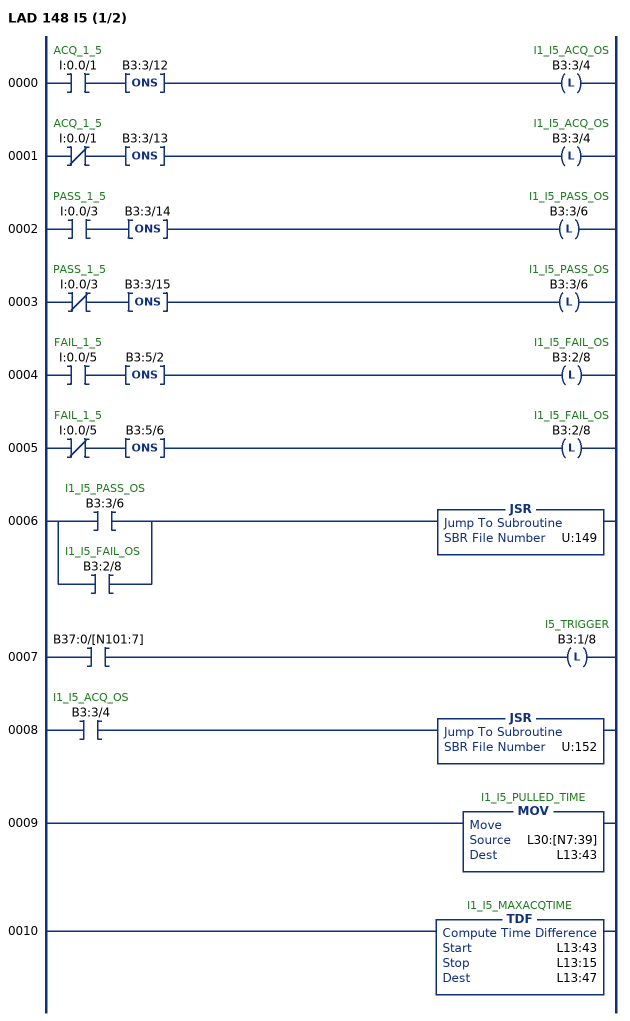
% Rung: 0 %
SOR XIC I:0.0/1 ONS B3:3/12 OTL B3:3/4 EOR
%   I:0.0/1  ACQ_1_5 %
%   B3:3/4  I1_I5_ACQ_OS %
% Rung: 1 %
SOR XIO I:0.0/1 ONS B3:3/13 OTL B3:3/4 EOR
%   I:0.0/1  ACQ_1_5 %
%   B3:3/4  I1_I5_ACQ_OS %
% Rung: 2 %
SOR XIC I:0.0/3 ONS B3:3/14 OTL B3:3/6 EOR
%   I:0.0/3  PASS_1_5 %
%   B3:3/6  I1_I5_PASS_OS %
% Rung: 3 %
SOR XIO I:0.0/3 ONS B3:3/15 OTL B3:3/6 EOR
%   I:0.0/3  PASS_1_5 %
%   B3:3/6  I1_I5_PASS_OS %
% Rung: 4 %
SOR XIC I:0.0/5 ONS B3:5/2 OTL B3:2/8 EOR
%   I:0.0/5  FAIL_1_5 %
%   B3:2/8  I1_I5_FAIL_OS %
% Rung: 5 %
SOR XIO I:0.0/5 ONS B3:5/6 OTL B3:2/8 EOR
%   I:0.0/5  FAIL_1_5 %
%   B3:2/8  I1_I5_FAIL_OS %
% Rung: 6 %
SOR BST XIC B3:3/6 NXB XIC B3:2/8 BND JSR U:149 EOR
%   B3:3/6  I1_I5_PASS_OS %
%   B3:2/8  I1_I5_FAIL_OS %
% Rung: 7 %
SOR XIC B37:0/[N101:7] OTL B3:1/8 EOR
%   B37:0  TOP_OK_1 %
%   N101:7  I5_TRIG_LOC %
%   B3:1/8  I5_TRIGGER %
% Rung: 8 %
SOR XIC B3:3/4 JSR U:152 EOR
%   B3:3/4  I1_I5_ACQ_OS %
% Rung: 9 %
SOR MOV L30:[N7:39] L13:43 EOR
%   N7:39  I5_OLDEST_PART_INDEX %
%   L13:43  I1_I5_PULLED_TIME %
% Rung: 10 %
SOR TDF L13:43 L13:15 L13:47 EOR
%   L13:43  I1_I5_PULLED_TIME %
%   L13:15  THE_TIME %
%   L13:47  I1_I5_MAXACQTIME %

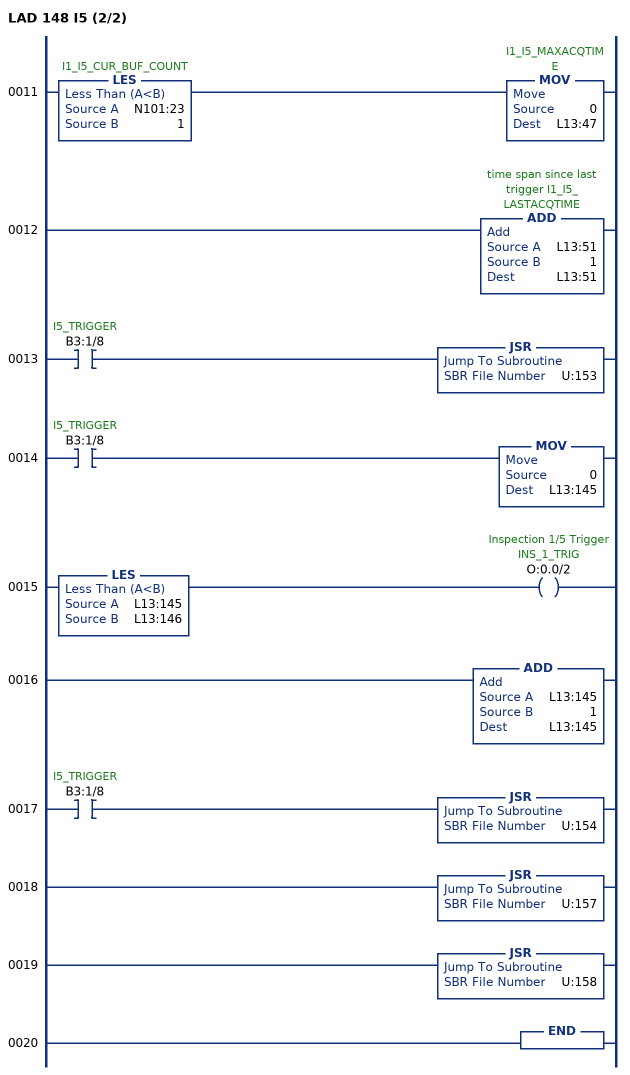
% Rung: 11 %
SOR LES N101:23 1 MOV 0 L13:47 EOR
%   N101:23  I1_I5_CUR_BUF_COUNT %
%   L13:47  I1_I5_MAXACQTIME %
% Rung: 12 %
SOR ADD L13:51 1 L13:51 EOR
%   L13:51  I1_I5_LASTACQTIME  "time span since last trigger" %
% Rung: 13 %
SOR XIC B3:1/8 JSR U:153 EOR
%   B3:1/8  I5_TRIGGER %
% Rung: 14 %
SOR XIC B3:1/8 MOV 0 L13:145 EOR
%   B3:1/8  I5_TRIGGER %
% Rung: 15 %
SOR LES L13:145 L13:146 OTE O:0.0/2 EOR
%   O:0.0/2  INS_1_TRIG  "Inspection 1/5 Trigger" %
% Rung: 16 %
SOR ADD L13:145 1 L13:145 EOR
% Rung: 17 %
SOR XIC B3:1/8 JSR U:154 EOR
%   B3:1/8  I5_TRIGGER %
% Rung: 18 %
SOR JSR U:157 EOR
% Rung: 19 %
SOR JSR U:158 EOR
% Rung: 20 %
SOR END EOR

LADDER 149 "I5 RESULT"
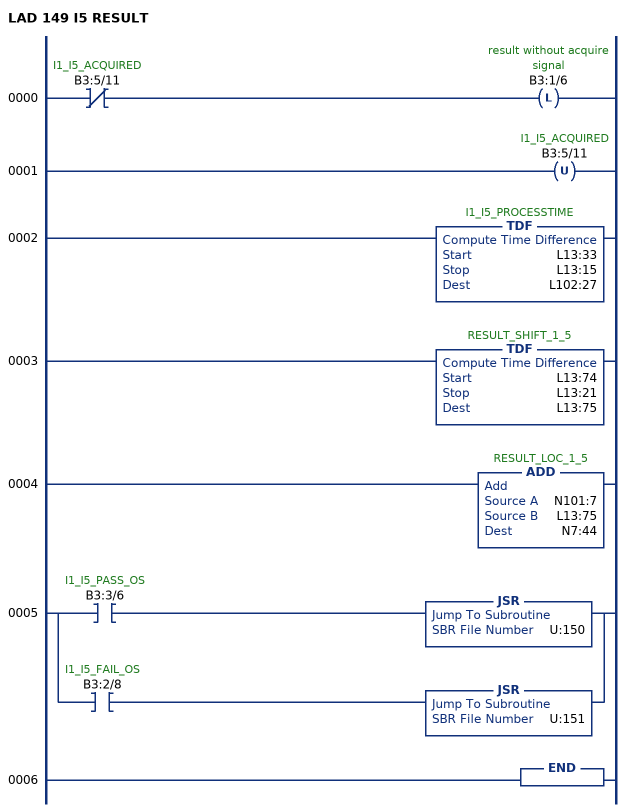
% Rung: 0 %
SOR XIO B3:5/11 OTL B3:1/6 EOR
%   B3:5/11  I1_I5_ACQUIRED %
%   B3:1/6  "result without acquire signal" %
% Rung: 1 %
SOR OTU B3:5/11 EOR
%   B3:5/11  I1_I5_ACQUIRED %
% Rung: 2 %
SOR TDF L13:33 L13:15 L102:27 EOR
%   L13:33  I1_I5_TIMEOFACQ %
%   L13:15  THE_TIME %
%   L102:27  I1_I5_PROCESSTIME %
% Rung: 3 %
SOR TDF L13:74 L13:21 L13:75 EOR
%   L13:74  I1_I5_PROC_START_POS %
%   L13:21  TOP_POSITION %
%   L13:75  RESULT_SHIFT_1_5 %
% Rung: 4 %
SOR ADD N101:7 L13:75 N7:44 EOR
%   N101:7  I5_TRIG_LOC %
%   L13:75  RESULT_SHIFT_1_5 %
%   N7:44  RESULT_LOC_1_5 %
% Rung: 5 %
SOR BST XIC B3:3/6 JSR U:150 NXB XIC B3:2/8 JSR U:151 BND EOR
%   B3:3/6  I1_I5_PASS_OS %
%   B3:2/8  I1_I5_FAIL_OS %
% Rung: 6 %
SOR END EOR

LADDER 150 "I5 PASS"
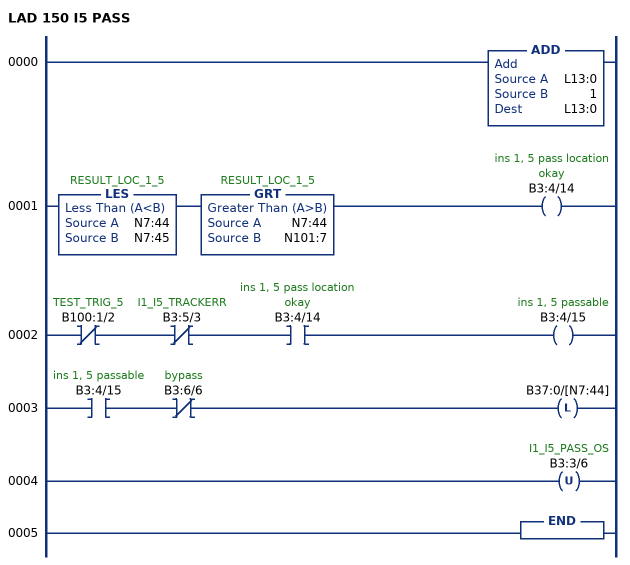
% Rung: 0 %
SOR ADD L13:0 1 L13:0 EOR
% Rung: 1 %
SOR LES N7:44 N7:45 GRT N7:44 N101:7 OTE B3:4/14 EOR
%   N7:44  RESULT_LOC_1_5 %
%   N7:45  I5_MAX_SHIFT  "ins 5 maximum result location" %
%   N101:7  I5_TRIG_LOC %
%   B3:4/14  "ins 1, 5 pass location okay" %
% Rung: 2 %
SOR XIO B100:1/2 XIO B3:5/3 XIC B3:4/14 OTE B3:4/15 EOR
%   B100:1/2  TEST_TRIG_5 %
%   B3:5/3  I1_I5_TRACKERR %
%   B3:4/14  "ins 1, 5 pass location okay" %
%   B3:4/15  "ins 1, 5 passable" %
% Rung: 3 %
SOR XIC B3:4/15 XIO B3:6/6 OTL B37:0/[N7:44] EOR
%   B3:4/15  "ins 1, 5 passable" %
%   B3:6/6  "bypass" %
%   B37:0  TOP_OK_1 %
%   N7:44  RESULT_LOC_1_5 %
% Rung: 4 %
SOR OTU B3:3/6 EOR
%   B3:3/6  I1_I5_PASS_OS %
% Rung: 5 %
SOR END EOR

LADDER 151 "I5 FAIL"
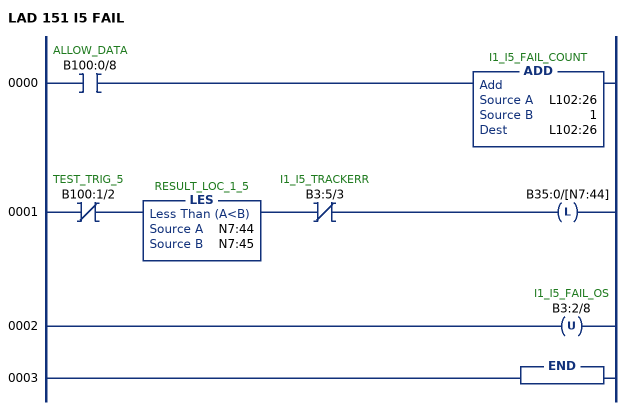
% Rung: 0 %
SOR XIC B100:0/8 ADD L102:26 1 L102:26 EOR
%   B100:0/8  ALLOW_DATA %
%   L102:26  I1_I5_FAIL_COUNT %
% Rung: 1 %
SOR XIO B100:1/2 LES N7:44 N7:45 XIO B3:5/3 OTL B35:0/[N7:44] EOR
%   B100:1/2  TEST_TRIG_5 %
%   N7:44  RESULT_LOC_1_5 %
%   N7:45  I5_MAX_SHIFT  "ins 5 maximum result location" %
%   B3:5/3  I1_I5_TRACKERR %
%   B35:0  TOP_NG %
% Rung: 2 %
SOR OTU B3:2/8 EOR
%   B3:2/8  I1_I5_FAIL_OS %
% Rung: 3 %
SOR END EOR

LADDER 152 "I5 ACQ"
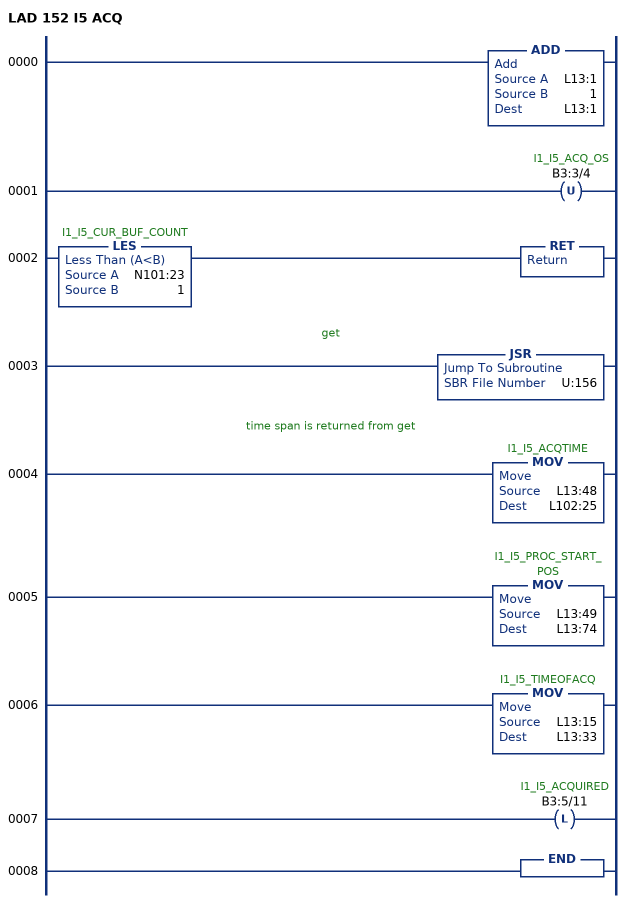
% Rung: 0 %
SOR ADD L13:1 1 L13:1 EOR
% Rung: 1 %
SOR OTU B3:3/4 EOR
%   B3:3/4  I1_I5_ACQ_OS %
% Rung: 2 %
SOR LES N101:23 1 RET EOR
%   N101:23  I1_I5_CUR_BUF_COUNT %
% Rung: 3 %
% get %
SOR JSR U:156 EOR
% Rung: 4 %
% time span is returned from get %
SOR MOV L13:48 L102:25 EOR
%   L13:48  I1_I5_TIME_SPAN %
%   L102:25  I1_I5_ACQTIME %
% Rung: 5 %
SOR MOV L13:49 L13:74 EOR
%   L13:49  I1_I5_PULLED_POS %
%   L13:74  I1_I5_PROC_START_POS %
% Rung: 6 %
SOR MOV L13:15 L13:33 EOR
%   L13:15  THE_TIME %
%   L13:33  I1_I5_TIMEOFACQ %
% Rung: 7 %
SOR OTL B3:5/11 EOR
%   B3:5/11  I1_I5_ACQUIRED %
% Rung: 8 %
SOR END EOR

LADDER 153 "I5 TESTER"
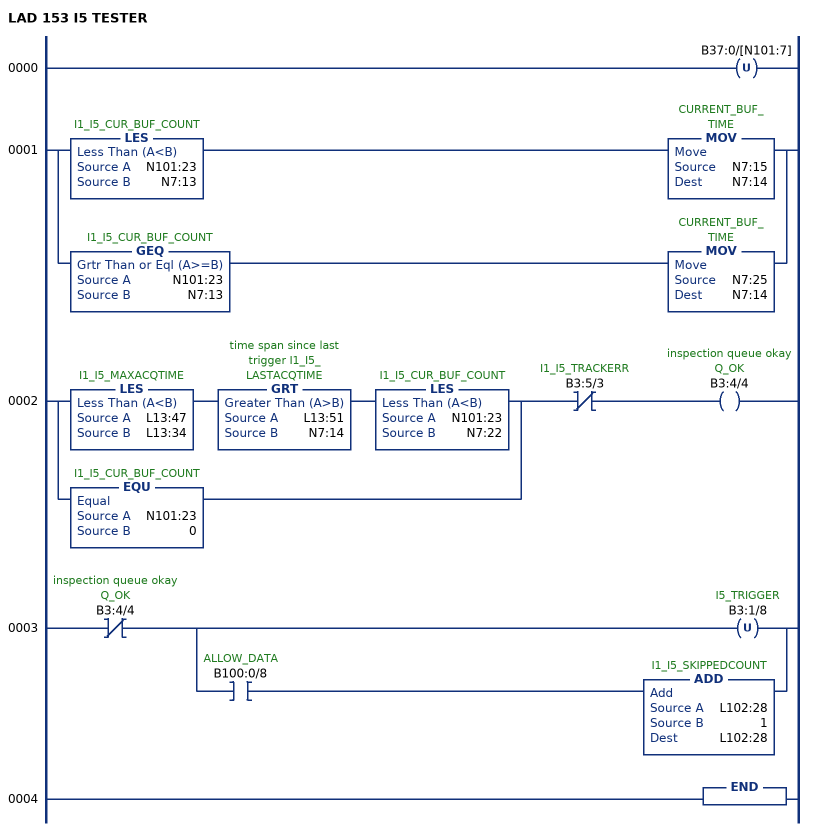
% Rung: 0 %
SOR OTU B37:0/[N101:7] EOR
%   B37:0  TOP_OK_1 %
%   N101:7  I5_TRIG_LOC %
% Rung: 1 %
SOR BST LES N101:23 N7:13 MOV N7:15 N7:14 NXB GEQ N101:23 N7:13 MOV N7:25 N7:14 BND EOR
%   N101:23  I1_I5_CUR_BUF_COUNT %
%   N7:13  BUF_TRANS  "cam to pc buf transition" %
%   N7:15  CAM_BUF_TIME  "cam buf time" %
%   N7:14  CURRENT_BUF_TIME %
%   N7:25  PC_BUF_TIME  "pc buf time" %
% Rung: 2 %
SOR BST LES L13:47 L13:34 GRT L13:51 N7:14 LES N101:23 N7:22 NXB EQU N101:23 0 BND XIO B3:5/3 OTE B3:4/4 EOR
%   L13:47  I1_I5_MAXACQTIME %
%   L13:34  MAX_ACQ_ALL  "absolute max acquire time before bypass trigger" %
%   L13:51  I1_I5_LASTACQTIME  "time span since last trigger" %
%   N7:14  CURRENT_BUF_TIME %
%   N101:23  I1_I5_CUR_BUF_COUNT %
%   N7:22  MAX_BUF_ALL  "max buffer count alowed before bypass" %
%   B3:5/3  I1_I5_TRACKERR %
%   B3:4/4  Q_OK  "inspection queue okay" %
% Rung: 3 %
SOR XIO B3:4/4 BST OTU B3:1/8 NXB XIC B100:0/8 ADD L102:28 1 L102:28 BND EOR
%   B3:4/4  Q_OK  "inspection queue okay" %
%   B3:1/8  I5_TRIGGER %
%   B100:0/8  ALLOW_DATA %
%   L102:28  I1_I5_SKIPPEDCOUNT %
% Rung: 4 %
SOR END EOR

LADDER 154 "I5 TRIG"
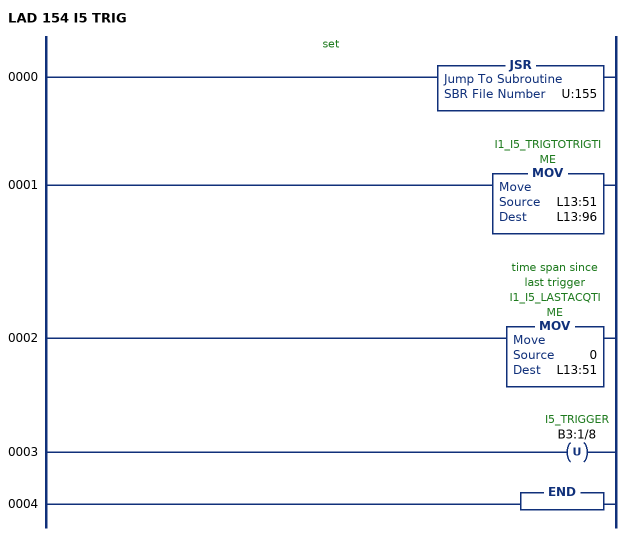
% Rung: 0 %
% set %
SOR JSR U:155 EOR
% Rung: 1 %
SOR MOV L13:51 L13:96 EOR
%   L13:51  I1_I5_LASTACQTIME  "time span since last trigger" %
%   L13:96  I1_I5_TRIGTOTRIGTIME %
% Rung: 2 %
SOR MOV 0 L13:51 EOR
%   L13:51  I1_I5_LASTACQTIME  "time span since last trigger" %
% Rung: 3 %
SOR OTU B3:1/8 EOR
%   B3:1/8  I5_TRIGGER %
% Rung: 4 %
SOR END EOR

LADDER 155 "I5 FIFOSET"
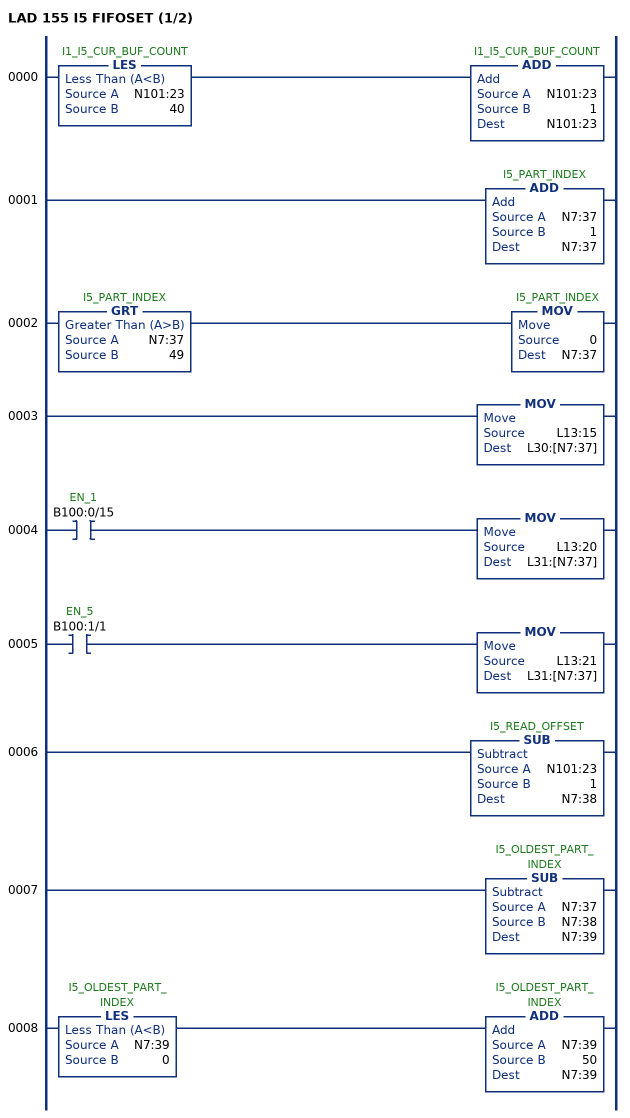
% Rung: 0 %
SOR LES N101:23 40 ADD N101:23 1 N101:23 EOR
%   N101:23  I1_I5_CUR_BUF_COUNT %
% Rung: 1 %
SOR ADD N7:37 1 N7:37 EOR
%   N7:37  I5_PART_INDEX %
% Rung: 2 %
SOR GRT N7:37 49 MOV 0 N7:37 EOR
%   N7:37  I5_PART_INDEX %
% Rung: 3 %
SOR MOV L13:15 L30:[N7:37] EOR
%   L13:15  THE_TIME %
%   N7:37  I5_PART_INDEX %
% Rung: 4 %
SOR XIC B100:0/15 MOV L13:20 L31:[N7:37] EOR
%   B100:0/15  EN_1 %
%   L13:20  BOT_POSITION %
%   N7:37  I5_PART_INDEX %
% Rung: 5 %
SOR XIC B100:1/1 MOV L13:21 L31:[N7:37] EOR
%   B100:1/1  EN_5 %
%   L13:21  TOP_POSITION %
%   N7:37  I5_PART_INDEX %
% Rung: 6 %
SOR SUB N101:23 1 N7:38 EOR
%   N101:23  I1_I5_CUR_BUF_COUNT %
%   N7:38  I5_READ_OFFSET %
% Rung: 7 %
SOR SUB N7:37 N7:38 N7:39 EOR
%   N7:37  I5_PART_INDEX %
%   N7:38  I5_READ_OFFSET %
%   N7:39  I5_OLDEST_PART_INDEX %
% Rung: 8 %
SOR LES N7:39 0 ADD N7:39 50 N7:39 EOR
%   N7:39  I5_OLDEST_PART_INDEX %

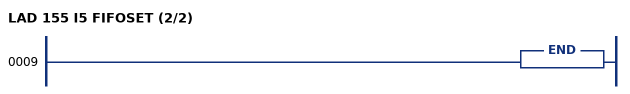
% Rung: 9 %
SOR END EOR

LADDER 156 "I5 FIFOGET"
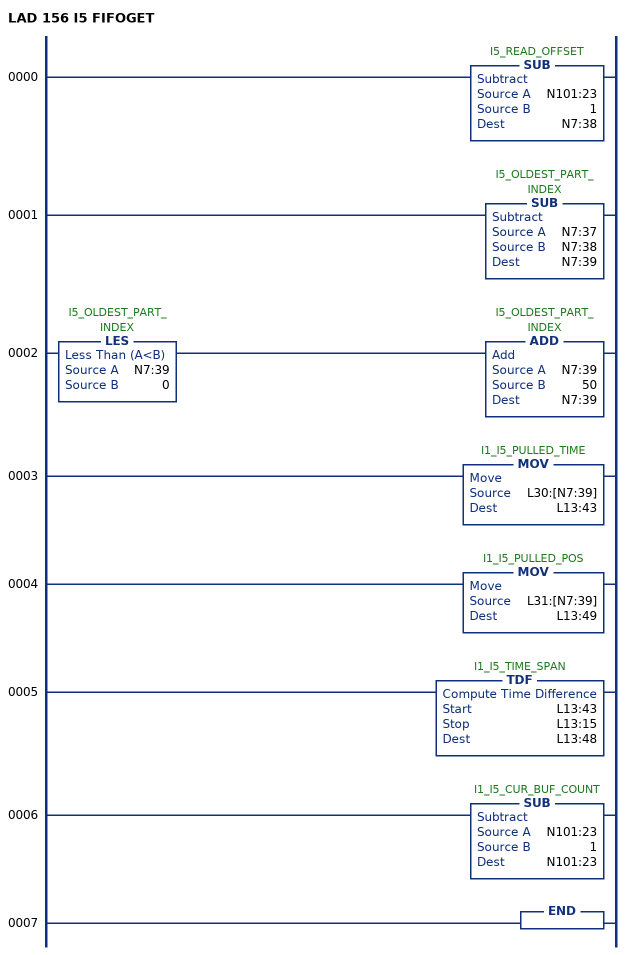
% Rung: 0 %
SOR SUB N101:23 1 N7:38 EOR
%   N101:23  I1_I5_CUR_BUF_COUNT %
%   N7:38  I5_READ_OFFSET %
% Rung: 1 %
SOR SUB N7:37 N7:38 N7:39 EOR
%   N7:37  I5_PART_INDEX %
%   N7:38  I5_READ_OFFSET %
%   N7:39  I5_OLDEST_PART_INDEX %
% Rung: 2 %
SOR LES N7:39 0 ADD N7:39 50 N7:39 EOR
%   N7:39  I5_OLDEST_PART_INDEX %
% Rung: 3 %
SOR MOV L30:[N7:39] L13:43 EOR
%   N7:39  I5_OLDEST_PART_INDEX %
%   L13:43  I1_I5_PULLED_TIME %
% Rung: 4 %
SOR MOV L31:[N7:39] L13:49 EOR
%   N7:39  I5_OLDEST_PART_INDEX %
%   L13:49  I1_I5_PULLED_POS %
% Rung: 5 %
SOR TDF L13:43 L13:15 L13:48 EOR
%   L13:43  I1_I5_PULLED_TIME %
%   L13:15  THE_TIME %
%   L13:48  I1_I5_TIME_SPAN %
% Rung: 6 %
SOR SUB N101:23 1 N101:23 EOR
%   N101:23  I1_I5_CUR_BUF_COUNT %
% Rung: 7 %
SOR END EOR

LADDER 157 "I5 DATA"
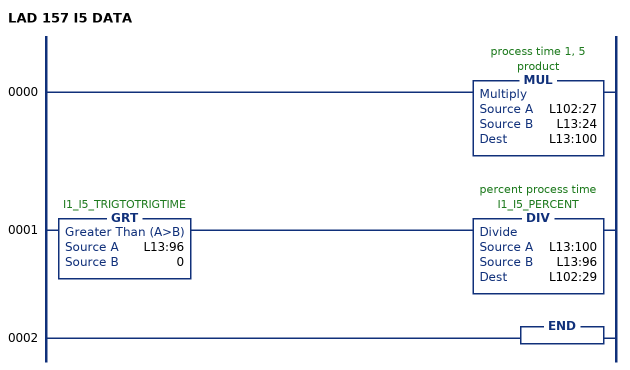
% Rung: 0 %
SOR MUL L102:27 L13:24 L13:100 EOR
%   L102:27  I1_I5_PROCESSTIME %
%   L13:24  "multiplyer to make devision come out to a percentage" %
%   L13:100  "process time 1, 5 product" %
% Rung: 1 %
SOR GRT L13:96 0 DIV L13:100 L13:96 L102:29 EOR
%   L13:96  I1_I5_TRIGTOTRIGTIME %
%   L13:100  "process time 1, 5 product" %
%   L102:29  I1_I5_PERCENT  "percent process time" %
% Rung: 2 %
SOR END EOR

LADDER 158 "I5 FAULT"
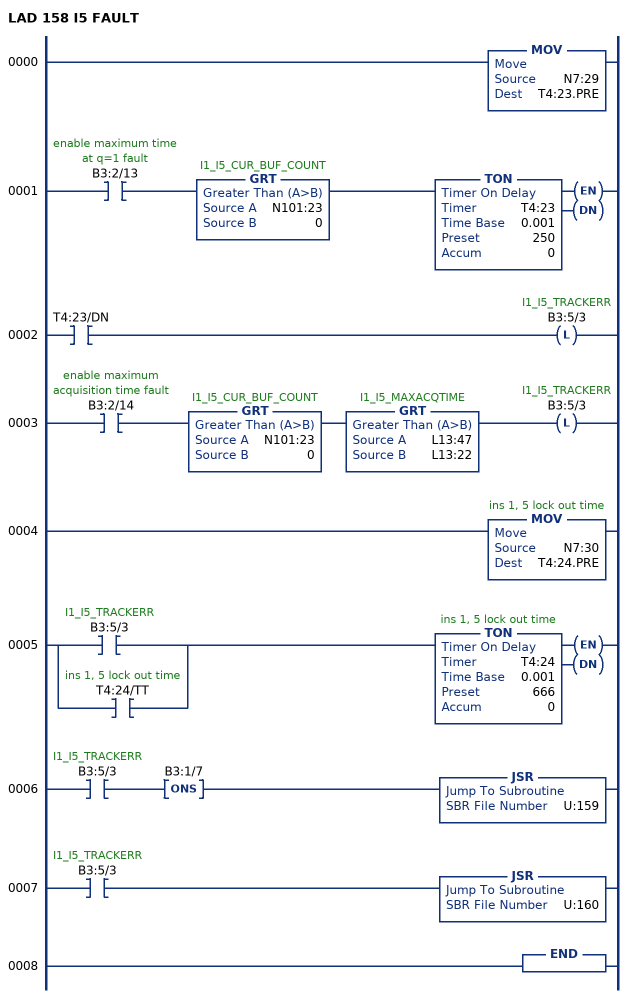
% Rung: 0 %
SOR MOV N7:29 T4:23.PRE EOR
%   N7:29  "max allowed ms time for q to be above 1 if safe fault is used" %
% Rung: 1 %
SOR XIC B3:2/13 GRT N101:23 0 TON T4:23 0.001 250 0 EOR
%   B3:2/13  "enable maximum time at q=1 fault" %
%   N101:23  I1_I5_CUR_BUF_COUNT %
% Rung: 2 %
SOR XIC T4:23/DN OTL B3:5/3 EOR
%   B3:5/3  I1_I5_TRACKERR %
% Rung: 3 %
SOR XIC B3:2/14 GRT N101:23 0 GRT L13:47 L13:22 OTL B3:5/3 EOR
%   B3:2/14  "enable maximum acquisition time fault" %
%   N101:23  I1_I5_CUR_BUF_COUNT %
%   L13:47  I1_I5_MAXACQTIME %
%   L13:22  "maximum of the longest acquire time allowed if maximum acquire time fault is enabled" %
%   B3:5/3  I1_I5_TRACKERR %
% Rung: 4 %
SOR MOV N7:30 T4:24.PRE EOR
%   N7:30  "ms time setting to lock out inspection to give all pending images a chance to clear" %
%   T4:24  "ins 1, 5 lock out time" %
% Rung: 5 %
SOR BST XIC B3:5/3 NXB XIC T4:24/TT BND TON T4:24 0.001 666 0 EOR
%   B3:5/3  I1_I5_TRACKERR %
%   T4:24  "ins 1, 5 lock out time" %
% Rung: 6 %
SOR XIC B3:5/3 ONS B3:1/7 JSR U:159 EOR
%   B3:5/3  I1_I5_TRACKERR %
% Rung: 7 %
SOR XIC B3:5/3 JSR U:160 EOR
%   B3:5/3  I1_I5_TRACKERR %
% Rung: 8 %
SOR END EOR

LADDER 159 "I5 FIX1"
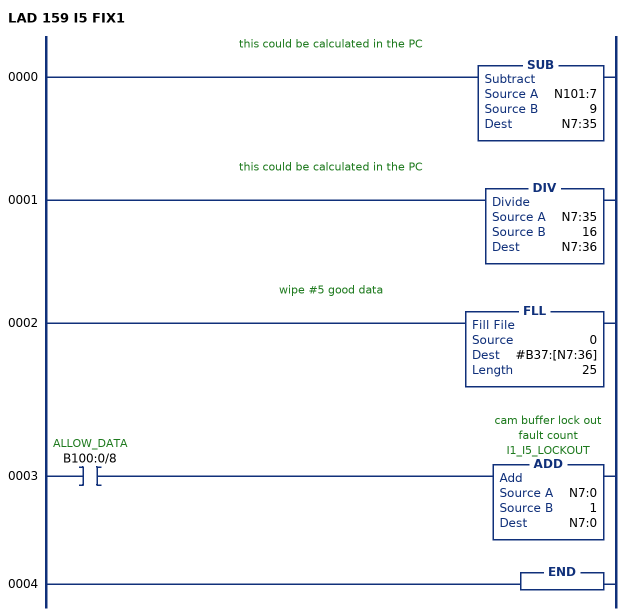
% Rung: 0 %
% this could be calculated in the PC %
SOR SUB N101:7 9 N7:35 EOR
%   N101:7  I5_TRIG_LOC %
% Rung: 1 %
% this could be calculated in the PC %
SOR DIV N7:35 16 N7:36 EOR
% Rung: 2 %
% wipe #5 good data %
SOR FLL 0 #B37:[N7:36] 25 EOR
% Rung: 3 %
SOR XIC B100:0/8 ADD N7:0 1 N7:0 EOR
%   B100:0/8  ALLOW_DATA %
%   N7:0  I1_I5_LOCKOUT  "cam buffer lock out fault count" %
% Rung: 4 %
SOR END EOR

LADDER 160 "I5 FIX2"
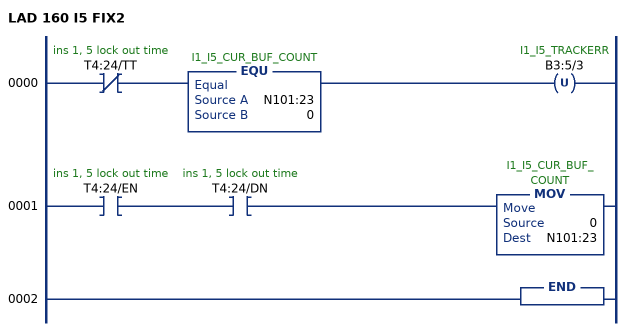
% Rung: 0 %
SOR XIO T4:24/TT EQU N101:23 0 OTU B3:5/3 EOR
%   T4:24  "ins 1, 5 lock out time" %
%   N101:23  I1_I5_CUR_BUF_COUNT %
%   B3:5/3  I1_I5_TRACKERR %
% Rung: 1 %
SOR XIC T4:24/EN XIC T4:24/DN MOV 0 N101:23 EOR
%   T4:24  "ins 1, 5 lock out time" %
%   N101:23  I1_I5_CUR_BUF_COUNT %
% Rung: 2 %
SOR END EOR

LADDER 161 "I6"
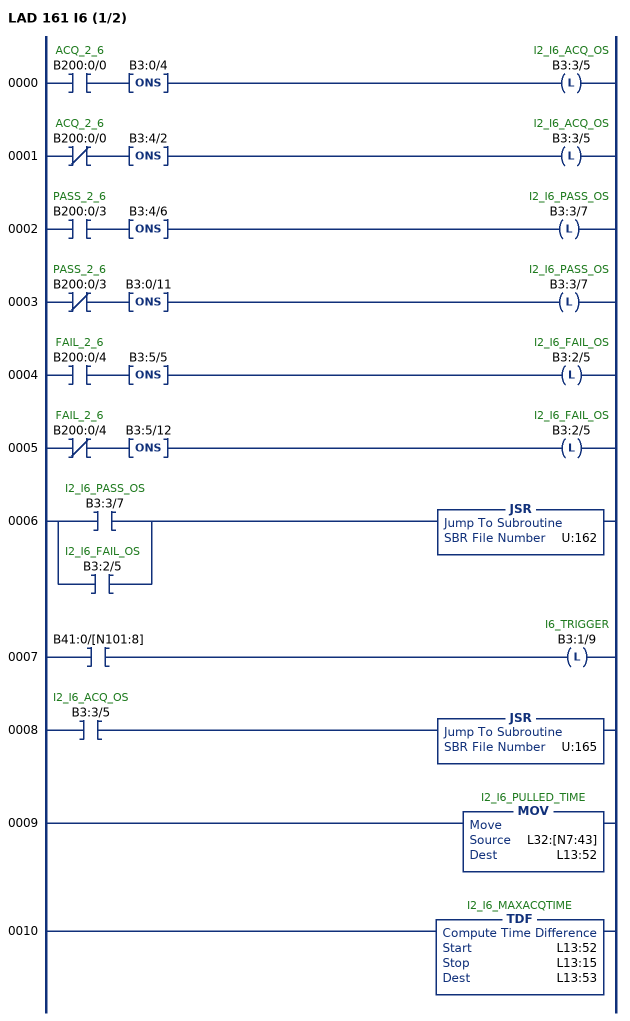
% Rung: 0 %
SOR XIC B200:0/0 ONS B3:0/4 OTL B3:3/5 EOR
%   B200:0/0  ACQ_2_6 %
%   B3:3/5  I2_I6_ACQ_OS %
% Rung: 1 %
SOR XIO B200:0/0 ONS B3:4/2 OTL B3:3/5 EOR
%   B200:0/0  ACQ_2_6 %
%   B3:3/5  I2_I6_ACQ_OS %
% Rung: 2 %
SOR XIC B200:0/3 ONS B3:4/6 OTL B3:3/7 EOR
%   B200:0/3  PASS_2_6 %
%   B3:3/7  I2_I6_PASS_OS %
% Rung: 3 %
SOR XIO B200:0/3 ONS B3:0/11 OTL B3:3/7 EOR
%   B200:0/3  PASS_2_6 %
%   B3:3/7  I2_I6_PASS_OS %
% Rung: 4 %
SOR XIC B200:0/4 ONS B3:5/5 OTL B3:2/5 EOR
%   B200:0/4  FAIL_2_6 %
%   B3:2/5  I2_I6_FAIL_OS %
% Rung: 5 %
SOR XIO B200:0/4 ONS B3:5/12 OTL B3:2/5 EOR
%   B200:0/4  FAIL_2_6 %
%   B3:2/5  I2_I6_FAIL_OS %
% Rung: 6 %
SOR BST XIC B3:3/7 NXB XIC B3:2/5 BND JSR U:162 EOR
%   B3:3/7  I2_I6_PASS_OS %
%   B3:2/5  I2_I6_FAIL_OS %
% Rung: 7 %
SOR XIC B41:0/[N101:8] OTL B3:1/9 EOR
%   B41:0  TOP_OK_3 %
%   N101:8  I6_TRIG_LOC %
%   B3:1/9  I6_TRIGGER %
% Rung: 8 %
SOR XIC B3:3/5 JSR U:165 EOR
%   B3:3/5  I2_I6_ACQ_OS %
% Rung: 9 %
SOR MOV L32:[N7:43] L13:52 EOR
%   N7:43  I6_OLDEST_PART_INDEX %
%   L13:52  I2_I6_PULLED_TIME %
% Rung: 10 %
SOR TDF L13:52 L13:15 L13:53 EOR
%   L13:52  I2_I6_PULLED_TIME %
%   L13:15  THE_TIME %
%   L13:53  I2_I6_MAXACQTIME %

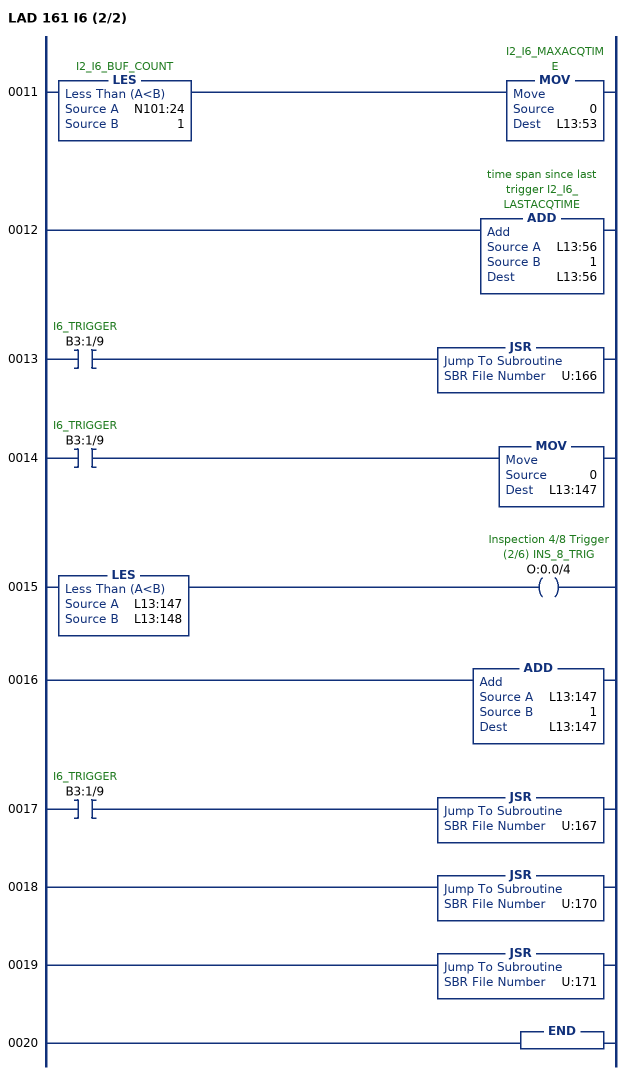
% Rung: 11 %
SOR LES N101:24 1 MOV 0 L13:53 EOR
%   N101:24  I2_I6_BUF_COUNT %
%   L13:53  I2_I6_MAXACQTIME %
% Rung: 12 %
SOR ADD L13:56 1 L13:56 EOR
%   L13:56  I2_I6_LASTACQTIME  "time span since last trigger" %
% Rung: 13 %
SOR XIC B3:1/9 JSR U:166 EOR
%   B3:1/9  I6_TRIGGER %
% Rung: 14 %
SOR XIC B3:1/9 MOV 0 L13:147 EOR
%   B3:1/9  I6_TRIGGER %
% Rung: 15 %
SOR LES L13:147 L13:148 OTE O:0.0/4 EOR
%   O:0.0/4  INS_8_TRIG  "Inspection 4/8 Trigger (2/6)" %
% Rung: 16 %
SOR ADD L13:147 1 L13:147 EOR
% Rung: 17 %
SOR XIC B3:1/9 JSR U:167 EOR
%   B3:1/9  I6_TRIGGER %
% Rung: 18 %
SOR JSR U:170 EOR
% Rung: 19 %
SOR JSR U:171 EOR
% Rung: 20 %
SOR END EOR

LADDER 162 "I6 RESULT"
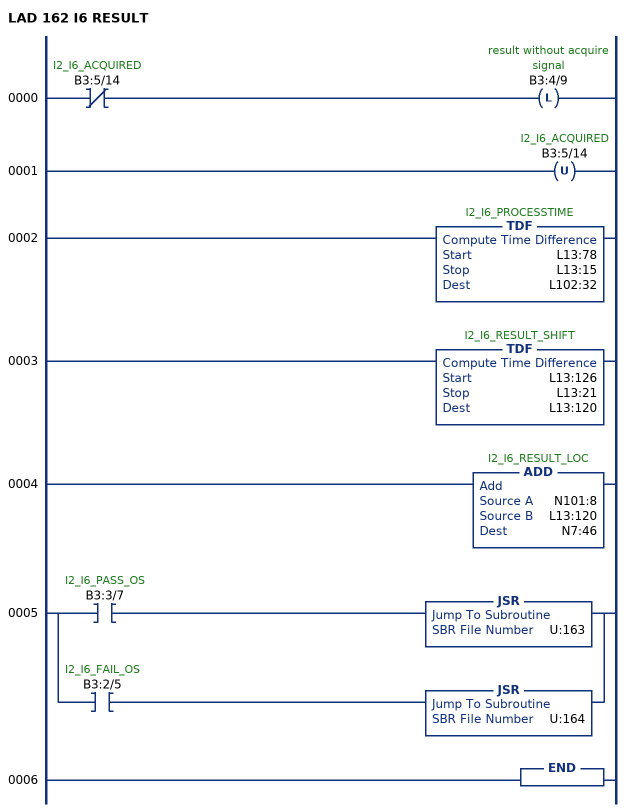
% Rung: 0 %
SOR XIO B3:5/14 OTL B3:4/9 EOR
%   B3:5/14  I2_I6_ACQUIRED %
%   B3:4/9  "result without acquire signal" %
% Rung: 1 %
SOR OTU B3:5/14 EOR
%   B3:5/14  I2_I6_ACQUIRED %
% Rung: 2 %
SOR TDF L13:78 L13:15 L102:32 EOR
%   L13:78  I2_I6_TIMEOFACQ %
%   L13:15  THE_TIME %
%   L102:32  I2_I6_PROCESSTIME %
% Rung: 3 %
SOR TDF L13:126 L13:21 L13:120 EOR
%   L13:126  I2_I6_PROC_START_POS %
%   L13:21  TOP_POSITION %
%   L13:120  I2_I6_RESULT_SHIFT %
% Rung: 4 %
SOR ADD N101:8 L13:120 N7:46 EOR
%   N101:8  I6_TRIG_LOC %
%   L13:120  I2_I6_RESULT_SHIFT %
%   N7:46  I2_I6_RESULT_LOC %
% Rung: 5 %
SOR BST XIC B3:3/7 JSR U:163 NXB XIC B3:2/5 JSR U:164 BND EOR
%   B3:3/7  I2_I6_PASS_OS %
%   B3:2/5  I2_I6_FAIL_OS %
% Rung: 6 %
SOR END EOR

LADDER 163 "I6 PASS"
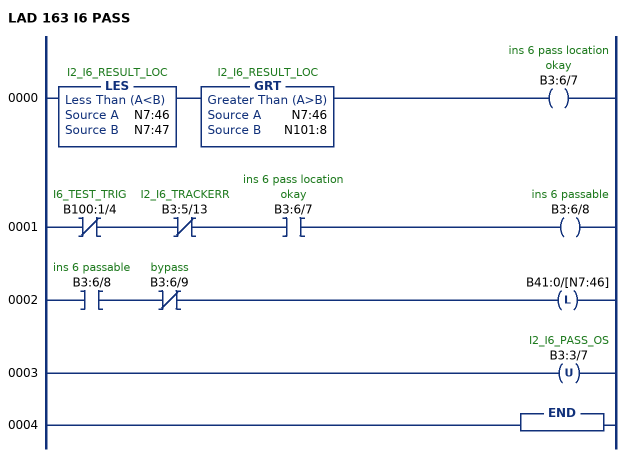
% Rung: 0 %
SOR LES N7:46 N7:47 GRT N7:46 N101:8 OTE B3:6/7 EOR
%   N7:46  I2_I6_RESULT_LOC %
%   N7:47  I6_MAX_SHIFT  "ins 6 maximum result location" %
%   N101:8  I6_TRIG_LOC %
%   B3:6/7  "ins 6 pass location okay" %
% Rung: 1 %
SOR XIO B100:1/4 XIO B3:5/13 XIC B3:6/7 OTE B3:6/8 EOR
%   B100:1/4  I6_TEST_TRIG %
%   B3:5/13  I2_I6_TRACKERR %
%   B3:6/7  "ins 6 pass location okay" %
%   B3:6/8  "ins 6 passable" %
% Rung: 2 %
SOR XIC B3:6/8 XIO B3:6/9 OTL B41:0/[N7:46] EOR
%   B3:6/8  "ins 6 passable" %
%   B3:6/9  "bypass" %
%   B41:0  TOP_OK_3 %
%   N7:46  I2_I6_RESULT_LOC %
% Rung: 3 %
SOR OTU B3:3/7 EOR
%   B3:3/7  I2_I6_PASS_OS %
% Rung: 4 %
SOR END EOR

LADDER 164 "I6 FAIL"
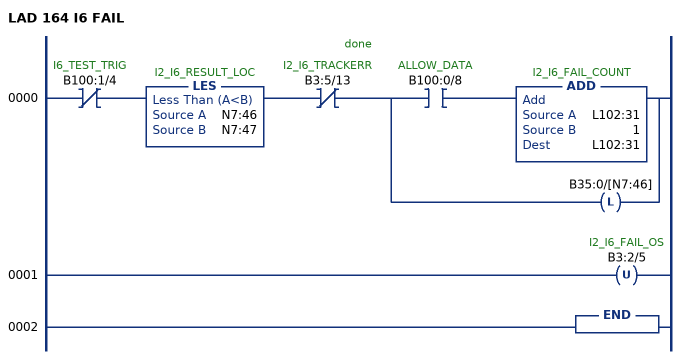
% Rung: 0 %
% done %
SOR XIO B100:1/4 LES N7:46 N7:47 XIO B3:5/13 BST XIC B100:0/8 ADD L102:31 1 L102:31 NXB OTL B35:0/[N7:46] BND EOR
%   B100:1/4  I6_TEST_TRIG %
%   N7:46  I2_I6_RESULT_LOC %
%   N7:47  I6_MAX_SHIFT  "ins 6 maximum result location" %
%   B3:5/13  I2_I6_TRACKERR %
%   B100:0/8  ALLOW_DATA %
%   L102:31  I2_I6_FAIL_COUNT %
%   B35:0  TOP_NG %
% Rung: 1 %
SOR OTU B3:2/5 EOR
%   B3:2/5  I2_I6_FAIL_OS %
% Rung: 2 %
SOR END EOR

LADDER 165 "I6 ACQ"
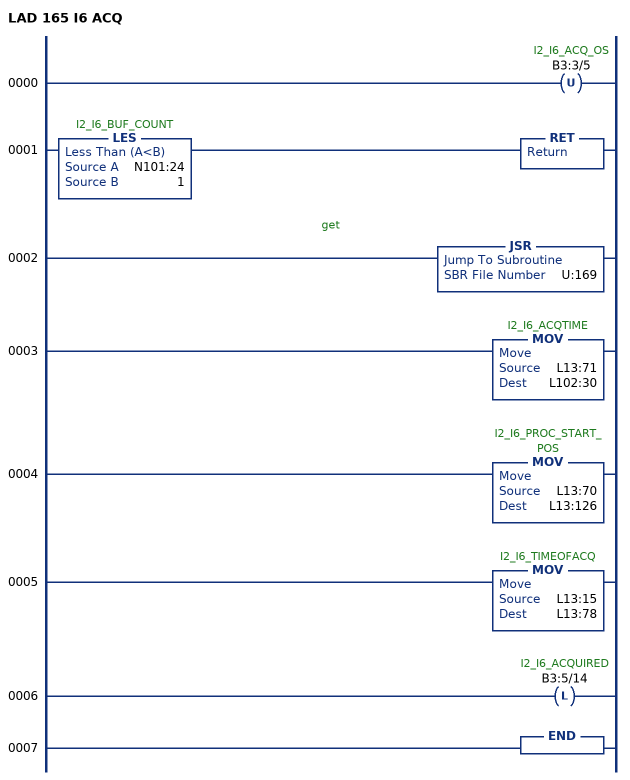
% Rung: 0 %
SOR OTU B3:3/5 EOR
%   B3:3/5  I2_I6_ACQ_OS %
% Rung: 1 %
SOR LES N101:24 1 RET EOR
%   N101:24  I2_I6_BUF_COUNT %
% Rung: 2 %
% get %
SOR JSR U:169 EOR
% Rung: 3 %
SOR MOV L13:71 L102:30 EOR
%   L13:71  I2_I6_TIME_SPAN %
%   L102:30  I2_I6_ACQTIME %
% Rung: 4 %
SOR MOV L13:70 L13:126 EOR
%   L13:70  I2_I6_PULLED_POS %
%   L13:126  I2_I6_PROC_START_POS %
% Rung: 5 %
SOR MOV L13:15 L13:78 EOR
%   L13:15  THE_TIME %
%   L13:78  I2_I6_TIMEOFACQ %
% Rung: 6 %
SOR OTL B3:5/14 EOR
%   B3:5/14  I2_I6_ACQUIRED %
% Rung: 7 %
SOR END EOR

LADDER 166 "I6 TESTER"
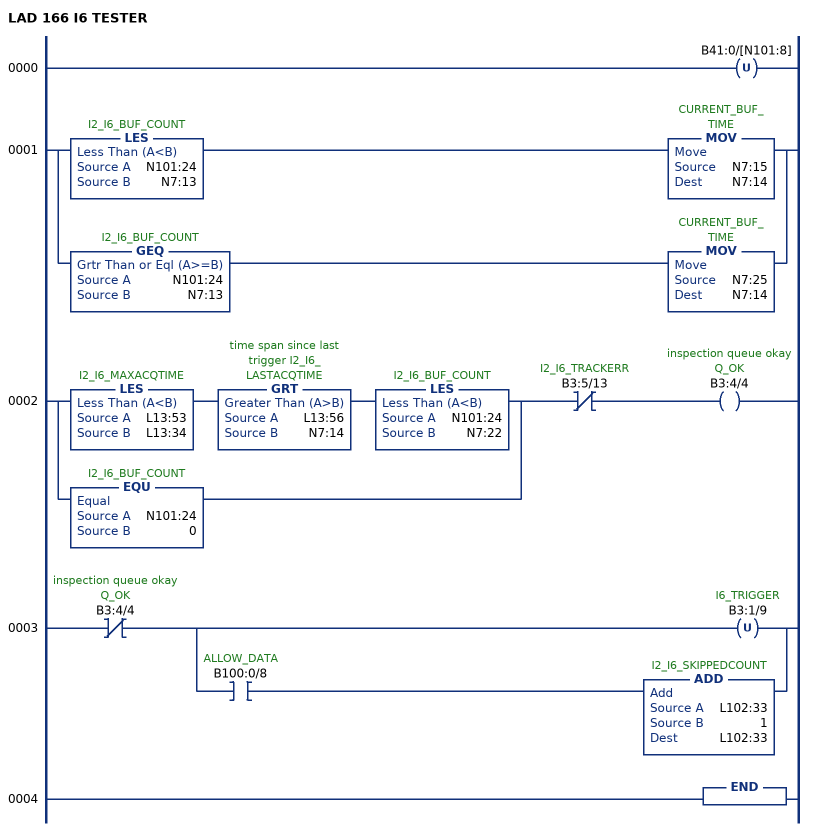
% Rung: 0 %
SOR OTU B41:0/[N101:8] EOR
%   B41:0  TOP_OK_3 %
%   N101:8  I6_TRIG_LOC %
% Rung: 1 %
SOR BST LES N101:24 N7:13 MOV N7:15 N7:14 NXB GEQ N101:24 N7:13 MOV N7:25 N7:14 BND EOR
%   N101:24  I2_I6_BUF_COUNT %
%   N7:13  BUF_TRANS  "cam to pc buf transition" %
%   N7:15  CAM_BUF_TIME  "cam buf time" %
%   N7:14  CURRENT_BUF_TIME %
%   N7:25  PC_BUF_TIME  "pc buf time" %
% Rung: 2 %
SOR BST LES L13:53 L13:34 GRT L13:56 N7:14 LES N101:24 N7:22 NXB EQU N101:24 0 BND XIO B3:5/13 OTE B3:4/4 EOR
%   L13:53  I2_I6_MAXACQTIME %
%   L13:34  MAX_ACQ_ALL  "absolute max acquire time before bypass trigger" %
%   L13:56  I2_I6_LASTACQTIME  "time span since last trigger" %
%   N7:14  CURRENT_BUF_TIME %
%   N101:24  I2_I6_BUF_COUNT %
%   N7:22  MAX_BUF_ALL  "max buffer count alowed before bypass" %
%   B3:5/13  I2_I6_TRACKERR %
%   B3:4/4  Q_OK  "inspection queue okay" %
% Rung: 3 %
SOR XIO B3:4/4 BST OTU B3:1/9 NXB XIC B100:0/8 ADD L102:33 1 L102:33 BND EOR
%   B3:4/4  Q_OK  "inspection queue okay" %
%   B3:1/9  I6_TRIGGER %
%   B100:0/8  ALLOW_DATA %
%   L102:33  I2_I6_SKIPPEDCOUNT %
% Rung: 4 %
SOR END EOR

LADDER 167 "I6 TRIG"
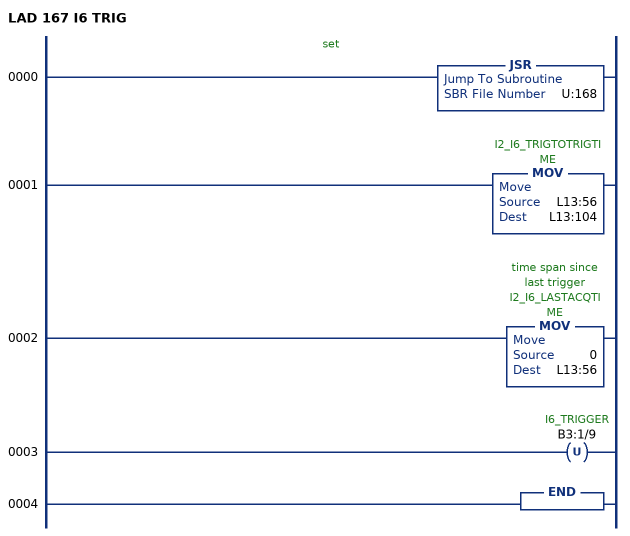
% Rung: 0 %
% set %
SOR JSR U:168 EOR
% Rung: 1 %
SOR MOV L13:56 L13:104 EOR
%   L13:56  I2_I6_LASTACQTIME  "time span since last trigger" %
%   L13:104  I2_I6_TRIGTOTRIGTIME %
% Rung: 2 %
SOR MOV 0 L13:56 EOR
%   L13:56  I2_I6_LASTACQTIME  "time span since last trigger" %
% Rung: 3 %
SOR OTU B3:1/9 EOR
%   B3:1/9  I6_TRIGGER %
% Rung: 4 %
SOR END EOR

LADDER 168 "I6 FIFOSET"
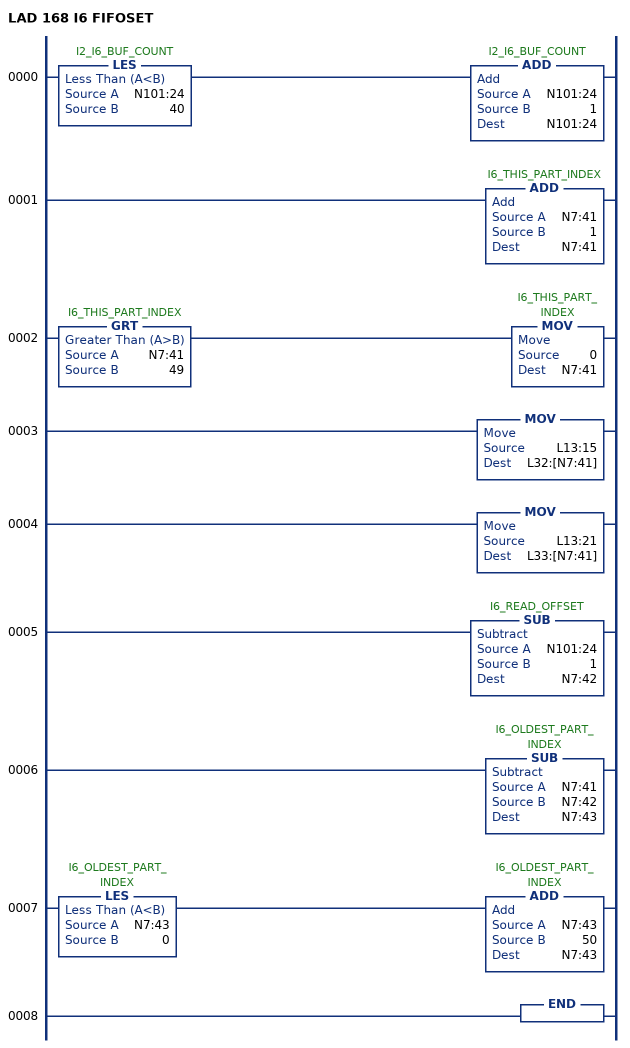
% Rung: 0 %
SOR LES N101:24 40 ADD N101:24 1 N101:24 EOR
%   N101:24  I2_I6_BUF_COUNT %
% Rung: 1 %
SOR ADD N7:41 1 N7:41 EOR
%   N7:41  I6_THIS_PART_INDEX %
% Rung: 2 %
SOR GRT N7:41 49 MOV 0 N7:41 EOR
%   N7:41  I6_THIS_PART_INDEX %
% Rung: 3 %
SOR MOV L13:15 L32:[N7:41] EOR
%   L13:15  THE_TIME %
%   N7:41  I6_THIS_PART_INDEX %
% Rung: 4 %
SOR MOV L13:21 L33:[N7:41] EOR
%   L13:21  TOP_POSITION %
%   N7:41  I6_THIS_PART_INDEX %
% Rung: 5 %
SOR SUB N101:24 1 N7:42 EOR
%   N101:24  I2_I6_BUF_COUNT %
%   N7:42  I6_READ_OFFSET %
% Rung: 6 %
SOR SUB N7:41 N7:42 N7:43 EOR
%   N7:41  I6_THIS_PART_INDEX %
%   N7:42  I6_READ_OFFSET %
%   N7:43  I6_OLDEST_PART_INDEX %
% Rung: 7 %
SOR LES N7:43 0 ADD N7:43 50 N7:43 EOR
%   N7:43  I6_OLDEST_PART_INDEX %
% Rung: 8 %
SOR END EOR

LADDER 169 "I6 FIFOGET"
